Staubli VAL3: cycle_isCallUse.pgx

program cycle_isCallUse()
  local num l_nResult
  local progItem l_pProg
begin
  // JUMP CALL USED
  if cycleStatus:bCALL
    do
      // reset the BIT
      cycleStatus:bCALL=false
      if cycleStatus:iToSuperV.sType=="PROG"
        // load the SUB PROG
        call prog:getProgItem(pProg,cycleStatus:iToSuperV.sData)
        // check it
        if pProg.sID!=""
          call cycle_run(pProg)
        else
          // STOP ALL
          cycleStatus:bToStop=true
        endIf
        // came back and restore
      else
        // just the LINE
        call cycle_doEvent(cycleStatus:iToSuperV,0)
      endIf
      // NESTED....
    until cycleStatus:bCALL==false
  endIf
end
